FUNCTION_BLOCK CommToMatlab (* Extracted Composite Function Block Type *)
  (* Version 5/20/2016, gulzha *)
  PACKAGE Main;
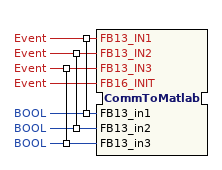
  EVENT_INPUT
    FB13_IN1 WITH FB13_in1; (* Normal Execution Request *)
    FB13_IN2 WITH FB13_in2;
    FB13_IN3 WITH FB13_in3;
    FB16_INIT; (* Initialization Request *)
  END_EVENT
  VAR_INPUT
    FB13_in1 : BOOL; (* Input event qualifier *)
    FB13_in2 : BOOL;
    FB13_in3 : BOOL;
  END_VAR
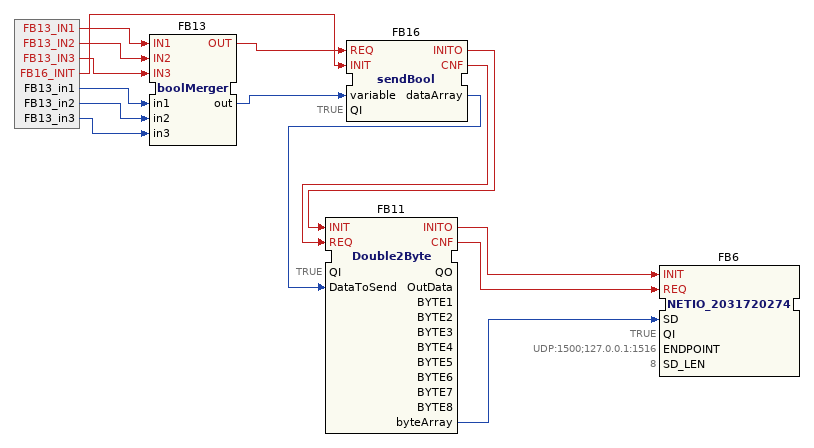
  FBS
    FB6 : NETIO_2031720274(QI := TRUE, ENDPOINT := UDP:1500;127.0.0.1:1516, SD_LEN := 8); {SET_ATTRIBUTE(Configuration.GenericFBType.InterfaceParams, Runtime.IoCommon#I:=1;SD:BYTE[8];RD:BYTE[8])}
    FB13 : boolMerger;
    FB16 : sendBool(QI := TRUE);
    FB11 : Double2Byte(QI := TRUE);
  END_FBS
  EVENT_CONNECTIONS
    FB13.OUT TO FB16.REQ;
    FB16.INITO TO FB11.INIT;
    FB11.INITO TO FB6.INIT;
    FB16.CNF TO FB11.REQ;
    FB11.CNF TO FB6.REQ;
    FB13_IN1 TO FB13.IN1;
    FB13_IN2 TO FB13.IN2;
    FB13_IN3 TO FB13.IN3;
    FB16_INIT TO FB16.INIT;
  END_CONNECTIONS
  DATA_CONNECTIONS
    FB13.out TO FB16.variable;
    FB11.byteArray TO FB6.SD;
    FB16.dataArray TO FB11.DataToSend;
    FB13_in1 TO FB13.in1;
    FB13_in2 TO FB13.in2;
    FB13_in3 TO FB13.in3;
  END_CONNECTIONS
END_FUNCTION_BLOCK
